PROGRAM P_Demo_FB_DALIV2Off
VAR
    fbFB_DALIV2Off        : FB_DALIV2Off;
    stCommandBuffer : ST_DALIV2CommandBuffer;

    bTrigger        : BOOL;
    nLampAddr        : BYTE := 0;


    bBusy           : BOOL;
    bErr            : BOOL;
    nErrId          : UDINT;
END_VAR

// =============================================================================
// 场景：消防联动：消防中心一键触发，PLC 广播本 FB 给整楼层所有非应急灯，瞬间关闭节能。...
//
// 价值：DALI 协议标准命令的轻量封装。
//
// 验证步骤：
//   1. 通信 FB 跑起；编译；登录。
//   2. 在线 bTrigger 一次上升沿；等 bBusy 回 FALSE。
//   3. 观察 short addr 0 灯的物理亮度变化是否符合本命令描述。
// =============================================================================
fbFB_DALIV2Off(
    bStart           := bTrigger,
    nAddr            := nLampAddr,
    eAddrType        := eDALIV2AddrTypeShort,
    eCommandPriority := eDALIV2CommandPriorityMiddle,
    stCommandBuffer  := stCommandBuffer
);

bBusy  := fbFB_DALIV2Off.bBusy;
bErr   := fbFB_DALIV2Off.bError;
nErrId := fbFB_DALIV2Off.nErrorId;

END_PROGRAM

(* stored: Version 1.1.0.1, ProductVersion 3.1.4024.5
   POU P_Demo_FB_DALIV2Off: Id {75735537-ad99-5a89-b918-c0d77419cd9d}, SpecialFunc None *)
